// SIMATIC S7-200 project (STEP 7-Micro/WIN), CPU 221 REL 01.10

ORGANIZATION_BLOCK MAIN:OB1
TITLE=PROGRAM COMMENTS
BEGIN
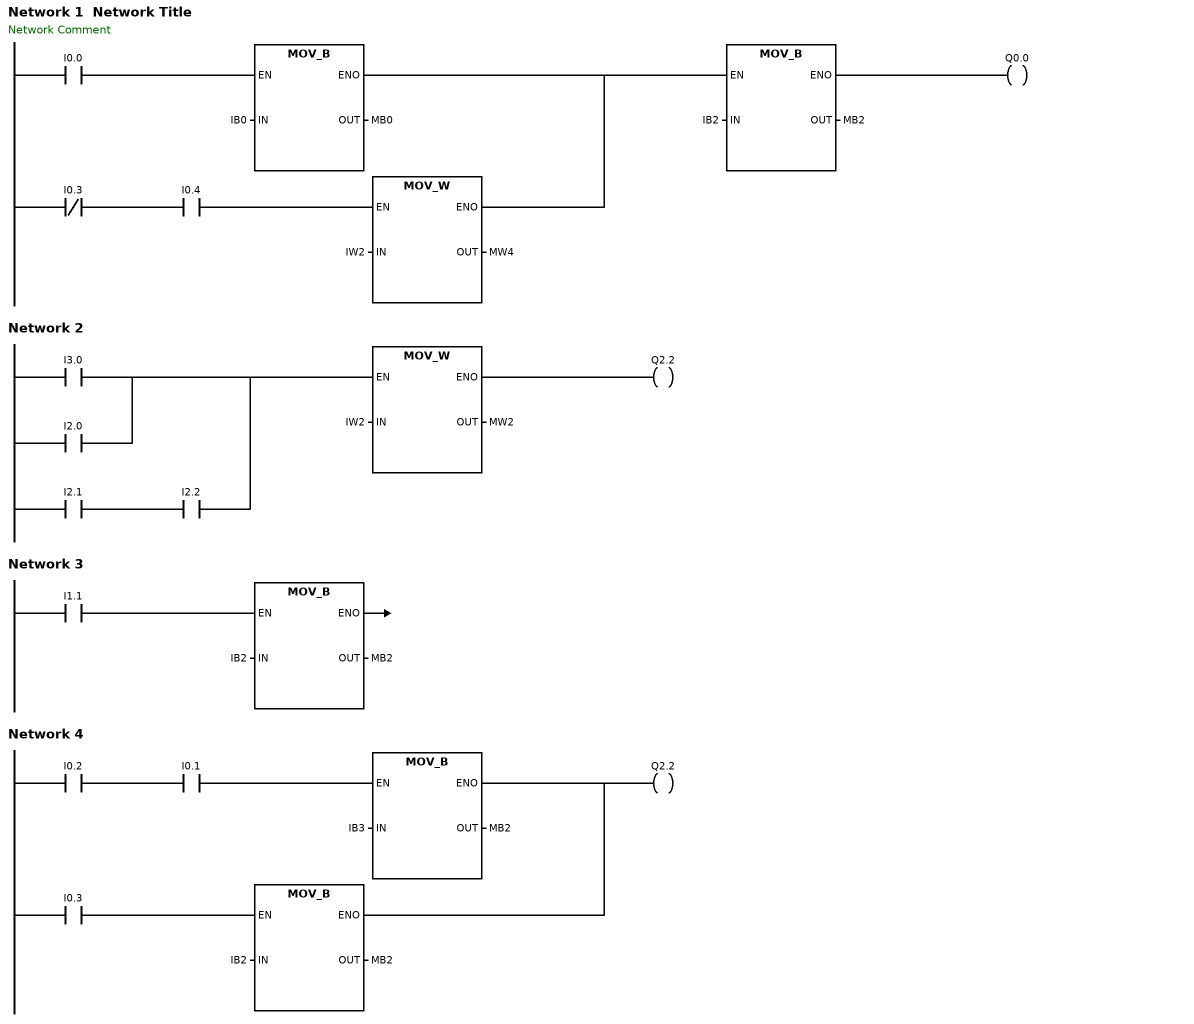
Network 1 // Network Title
// Network Comment
LD     I0.0
MOVB   IB0, MB0
AENO
LDN    I0.3
A      I0.4
MOVW   IW2, MW4
AENO
OLD
MOVB   IB2, MB2
AENO
=      Q0.0
Network 2
LD     I3.0
O      I2.0
LD     I2.1
A      I2.2
OLD
MOVW   IW2, MW2
AENO
=      Q2.2
Network 3
LD     I1.1
MOVB   IB2, MB2
Network 4
LD     I0.2
A      I0.1
MOVB   IB3, MB2
AENO
LD     I0.3
MOVB   IB2, MB2
AENO
OLD
=      Q2.2
END_ORGANIZATION_BLOCK
